FUNCTION_BLOCK FB_LoggerTest EXTENDS TcUnit.FB_TestSuite
VAR

END_VAR


T01_TestDodawaniaZgloszen ();
T02_TestDodawaniaZgloszen2 ();
T03_TestDodawaniaZgloszen3 ();

METHOD PRIVATE T01_TestDodawaniaZgloszen
VAR
	sttmpEvent: ST_BaseEvents_RowInQueue;
END_VAR
IF (TcUnit.TEST_ORDERED ('T01_TestDodawaniaZgloszen')) THEN
	WRITE_PROTECTED_BOOL (Ptr := ADR (GVL.fbLogger.bClearMemory), Value := TRUE);
	GVL.fbLogger ();
	AssertEquals_INT (Expected := 0, Actual := GVL.fbLogger.stBuffer.iNumerOfEvents, 	Message := 'T01a - bledna ilosc w kolejce');
	AssertEquals_INT (Expected := 0, Actual := GVL.fbLogger.stmemory.iNumberOfRow,		Message := 'T01b - bledna ilosc zgloszen');
//wyslanie zgloszenia 
	sttmpEvent.bActive				:= TRUE;
	sttmpEvent.bConfirm				:= TRUE;
	sttmpEvent.bIgnoreRepetitions	:= TRUE;
	sttmpEvent.dtStart				:= DT#2025-09-25-01:00:00;
	sttmpEvent.eEventCategory		:= E_BaseEvents_Category.Error;
	sttmpEvent.eEventAction			:= E_BaseEvents_Action.Start;
	sttmpEvent.uiIDEvent			:= 1;
	sttmpEvent.uiIDItem				:= 2;
	GVL.fbLogger.ReportEvent (stEvent := sttmpEvent);
	AssertEquals_INT (Expected := 1, Actual := GVL.fbLogger.stBuffer.iNumerOfEvents, 	Message := 'T02a - bledna ilosc w kolejce');
	AssertEquals_INT (Expected := 0, Actual := GVL.fbLogger.stmemory.iNumberOfRow,		Message := 'T02b - bledna ilosc zgloszen');
	GVL.fbLogger ();
	AssertEquals_INT (Expected := 0, Actual := GVL.fbLogger.stBuffer.iNumerOfEvents, 					Message := 'T03a - bledna ilosc w kolejce');
	AssertEquals_INT (Expected := 1, Actual := GVL.fbLogger.stmemory.iNumberOfRow,						Message := 'T03b - bledna ilosc zgloszen');
	AssertEquals_INT (Expected := 1, Actual := GVL.fbLogger.stNumberOfReports.iNumberOfActive,			Message := 'T03c - bledna ilosc zgloszen');
	AssertTrue (Condition := GVL.fbLogger.stNumberOfReports.arrActive [E_BaseEvents_Category.Error],	Message := 'T03d - bledny stan');
	AssertFalse (Condition := GVL.fbLogger.stNumberOfReports.arrActive [E_BaseEvents_Category.Alarm],	Message := 'T03d - bledny stan');
	AssertTrue (Condition := GVL.fbLogger.stNumberOfReports.bIsActive,									Message := 'T03e - bledny stan');
	AssertEquals_INT (Expected := 1, Actual := GVL.fbLogger.stNumberOfReports.iTotalNumer,				Message := 'T03f - bledna ilosc zgloszen');
//potwierdzenie zgloszenia 
	sttmpEvent.eEventAction			:= E_BaseEvents_Action.Confirm;
	sttmpEvent.uiIDEvent			:= 1;
	sttmpEvent.uiIDItem				:= 2;
	sttmpEvent.dtConfirmed			:= DT#2025-09-25-01:01:00;
	GVL.fbLogger.ReportEvent (stEvent := sttmpEvent);
	AssertEquals_INT (Expected := 1, Actual := GVL.fbLogger.stBuffer.iNumerOfEvents, 					Message := 'T04a - bledna ilosc w kolejce');
	AssertEquals_INT (Expected := 1, Actual := GVL.fbLogger.stmemory.iNumberOfRow,						Message := 'T04b - bledna ilosc zgloszen');
	GVL.fbLogger ();
	AssertEquals_INT (Expected := 0, Actual := GVL.fbLogger.stBuffer.iNumerOfEvents, 					Message := 'T05a - bledna ilosc w kolejce');
	AssertEquals_INT (Expected := 1, Actual := GVL.fbLogger.stmemory.iNumberOfRow,						Message := 'T05b - bledna ilosc zgloszen');
	AssertEquals_INT (Expected := 1, Actual := GVL.fbLogger.stNumberOfReports.iNumberOfActive,			Message := 'T05c - bledna ilosc zgloszen');
	AssertTrue (Condition := GVL.fbLogger.stNumberOfReports.arrActive [E_BaseEvents_Category.Error],	Message := 'T05d - bledny stan');
	AssertFalse (Condition := GVL.fbLogger.stNumberOfReports.arrActive [E_BaseEvents_Category.Alarm],	Message := 'T05d - bledny stan');
	AssertTrue (Condition := GVL.fbLogger.stNumberOfReports.bIsActive,									Message := 'T05e - bledny stan');
	AssertEquals_INT (Expected := 1, Actual := GVL.fbLogger.stNumberOfReports.iTotalNumer,				Message := 'T05f - bledna ilosc zgloszen');
//zamkniecie zgloszenia 
	sttmpEvent.eEventAction			:= E_BaseEvents_Action.Stop;
	sttmpEvent.uiIDEvent			:= 1;
	sttmpEvent.uiIDItem				:= 2;
	sttmpEvent.dtFinish				:= DT#2025-09-25-01:02:00;
	GVL.fbLogger.ReportEvent (stEvent := sttmpEvent);
	AssertEquals_INT (Expected := 1, Actual := GVL.fbLogger.stBuffer.iNumerOfEvents, 					Message := 'T04a - bledna ilosc w kolejce');
	AssertEquals_INT (Expected := 1, Actual := GVL.fbLogger.stmemory.iNumberOfRow,						Message := 'T04b - bledna ilosc zgloszen');
	GVL.fbLogger ();
	AssertEquals_INT (Expected := 0, Actual := GVL.fbLogger.stBuffer.iNumerOfEvents, 					Message := 'T05a - bledna ilosc w kolejce');
	AssertEquals_INT (Expected := 1, Actual := GVL.fbLogger.stmemory.iNumberOfRow,						Message := 'T05b - bledna ilosc zgloszen');
	AssertEquals_INT (Expected := 0, Actual := GVL.fbLogger.stNumberOfReports.iNumberOfActive,			Message := 'T05c - bledna ilosc zgloszen');
	AssertFalse (Condition := GVL.fbLogger.stNumberOfReports.arrActive [E_BaseEvents_Category.Error],	Message := 'T05d - bledny stan');
	AssertFalse (Condition := GVL.fbLogger.stNumberOfReports.arrActive [E_BaseEvents_Category.Alarm],	Message := 'T05d - bledny stan');
	Assertfalse (Condition := GVL.fbLogger.stNumberOfReports.bIsActive,									Message := 'T05e - bledny stan');
	AssertEquals_INT (Expected := 1, Actual := GVL.fbLogger.stNumberOfReports.iTotalNumer,				Message := 'T05f - bledna ilosc zgloszen');
	
	
	TcUnit.TEST_FINISHED ();
END_IF
END_METHOD

METHOD PRIVATE T02_TestDodawaniaZgloszen2
VAR
	sttmpEvent: ST_BaseEvents_RowInQueue;
END_VAR
IF (TcUnit.TEST_ORDERED ('T02_TestDodawaniaZgloszen2')) THEN
	GVL.fbLogger ();
	AssertEquals_INT (Expected := 0, Actual := GVL.fbLogger.stBuffer.iNumerOfEvents, 	Message := 'T01a - bledna ilosc w kolejce');
	AssertEquals_INT (Expected := 1, Actual := GVL.fbLogger.stmemory.iNumberOfRow,		Message := 'T01b - bledna ilosc zgloszen');
//wyslanie zgloszenia 
	sttmpEvent.bActive				:= TRUE;
	sttmpEvent.bConfirm				:= TRUE;
	sttmpEvent.bIgnoreRepetitions	:= TRUE;
	sttmpEvent.dtStart				:= DT#2025-09-25-02:00:00;
	sttmpEvent.eEventCategory		:= E_BaseEvents_Category.Error;
	sttmpEvent.eEventAction			:= E_BaseEvents_Action.Start;
	sttmpEvent.uiIDEvent			:= 1;
	sttmpEvent.uiIDItem				:= 2;
	GVL.fbLogger.ReportEvent (stEvent := sttmpEvent);
	AssertEquals_INT (Expected := 1, Actual := GVL.fbLogger.stBuffer.iNumerOfEvents, 					Message := 'T02a - bledna ilosc w kolejce');
	AssertEquals_INT (Expected := 1, Actual := GVL.fbLogger.stmemory.iNumberOfRow,						Message := 'T02b - bledna ilosc zgloszen');
	GVL.fbLogger ();
	AssertEquals_INT (Expected := 0, Actual := GVL.fbLogger.stBuffer.iNumerOfEvents, 					Message := 'T03a - bledna ilosc w kolejce');
	AssertEquals_INT (Expected := 2, Actual := GVL.fbLogger.stmemory.iNumberOfRow,						Message := 'T03b - bledna ilosc zgloszen');
	AssertEquals_INT (Expected := 1, Actual := GVL.fbLogger.stNumberOfReports.iNumberOfActive,			Message := 'T03c - bledna ilosc zgloszen');
	AssertTrue (Condition := GVL.fbLogger.stNumberOfReports.arrActive [E_BaseEvents_Category.Error],	Message := 'T03d - bledny stan');
	AssertFalse (Condition := GVL.fbLogger.stNumberOfReports.arrActive [E_BaseEvents_Category.Alarm],	Message := 'T03d - bledny stan');
	AssertTrue (Condition := GVL.fbLogger.stNumberOfReports.bIsActive,									Message := 'T03e - bledny stan');
	AssertEquals_INT (Expected := 2, Actual := GVL.fbLogger.stNumberOfReports.iTotalNumer,				Message := 'T03f - bledna ilosc zgloszen');
//zamkniecie zgloszenia  bez potwierdzenia a wymagane nic się nei powinno stać
	sttmpEvent.eEventAction			:= E_BaseEvents_Action.Stop;
	sttmpEvent.uiIDEvent			:= 1;
	sttmpEvent.uiIDItem				:= 2;
	sttmpEvent.dtFinish				:= DT#2025-09-25-02:00:00;
	GVL.fbLogger.ReportEvent (stEvent := sttmpEvent);
	AssertEquals_INT (Expected := 1, Actual := GVL.fbLogger.stBuffer.iNumerOfEvents, 					Message := 'T04a - bledna ilosc w kolejce');
	AssertEquals_INT (Expected := 2, Actual := GVL.fbLogger.stmemory.iNumberOfRow,						Message := 'T04b - bledna ilosc zgloszen');
	GVL.fbLogger ();
	AssertEquals_INT (Expected := 0, Actual := GVL.fbLogger.stBuffer.iNumerOfEvents, 					Message := 'T05a - bledna ilosc w kolejce');
	AssertEquals_INT (Expected := 2, Actual := GVL.fbLogger.stmemory.iNumberOfRow,						Message := 'T05b - bledna ilosc zgloszen');
	AssertEquals_INT (Expected := 1, Actual := GVL.fbLogger.stNumberOfReports.iNumberOfActive,			Message := 'T05c - bledna ilosc zgloszen');
	AssertTrue (Condition := GVL.fbLogger.stNumberOfReports.arrActive [E_BaseEvents_Category.Error],	Message := 'T05d - bledny stan');
	AssertFalse (Condition := GVL.fbLogger.stNumberOfReports.arrActive [E_BaseEvents_Category.Alarm],	Message := 'T05d - bledny stan');
	AssertTrue (Condition := GVL.fbLogger.stNumberOfReports.bIsActive,									Message := 'T05e - bledny stan');
	AssertEquals_INT (Expected := 2, Actual := GVL.fbLogger.stNumberOfReports.iTotalNumer,				Message := 'T05f - bledna ilosc zgloszen');
//potwierdzenie zgloszenia 
	sttmpEvent.eEventAction			:= E_BaseEvents_Action.Confirm;
	sttmpEvent.uiIDEvent			:= 1;
	sttmpEvent.uiIDItem				:= 2;
	sttmpEvent.dtConfirmed			:= DT#2025-09-25-02:01:00;
	GVL.fbLogger.ReportEvent (stEvent := sttmpEvent);
	AssertEquals_INT (Expected := 1, Actual := GVL.fbLogger.stBuffer.iNumerOfEvents, 					Message := 'T06a - bledna ilosc w kolejce');
	AssertEquals_INT (Expected := 2, Actual := GVL.fbLogger.stmemory.iNumberOfRow,						Message := 'T06b - bledna ilosc zgloszen');
	GVL.fbLogger ();
	AssertEquals_INT (Expected := 0, Actual := GVL.fbLogger.stBuffer.iNumerOfEvents, 					Message := 'T07a - bledna ilosc w kolejce');
	AssertEquals_INT (Expected := 2, Actual := GVL.fbLogger.stmemory.iNumberOfRow,						Message := 'T07b - bledna ilosc zgloszen');
	AssertEquals_INT (Expected := 1, Actual := GVL.fbLogger.stNumberOfReports.iNumberOfActive,			Message := 'T07c - bledna ilosc zgloszen');
	AssertTrue (Condition := GVL.fbLogger.stNumberOfReports.arrActive [E_BaseEvents_Category.Error],	Message := 'T07d - bledny stan');
	AssertFalse (Condition := GVL.fbLogger.stNumberOfReports.arrActive [E_BaseEvents_Category.Alarm],	Message := 'T07d - bledny stan');
	AssertTrue (Condition := GVL.fbLogger.stNumberOfReports.bIsActive,									Message := 'T07e - bledny stan');
	AssertEquals_INT (Expected := 2, Actual := GVL.fbLogger.stNumberOfReports.iTotalNumer,				Message := 'T07f - bledna ilosc zgloszen');
//zamkniecie zgloszenia 
	sttmpEvent.eEventAction			:= E_BaseEvents_Action.Stop;
	sttmpEvent.uiIDEvent			:= 1;
	sttmpEvent.uiIDItem				:= 2;
	sttmpEvent.dtFinish				:= DT#2025-09-25-02:02:00;
	GVL.fbLogger.ReportEvent (stEvent := sttmpEvent);
	AssertEquals_INT (Expected := 1, Actual := GVL.fbLogger.stBuffer.iNumerOfEvents, 					Message := 'T08a - bledna ilosc w kolejce');
	AssertEquals_INT (Expected := 2, Actual := GVL.fbLogger.stmemory.iNumberOfRow,						Message := 'T08b - bledna ilosc zgloszen');
	GVL.fbLogger ();
	AssertEquals_INT (Expected := 0, Actual := GVL.fbLogger.stBuffer.iNumerOfEvents, 					Message := 'T09a - bledna ilosc w kolejce');
	AssertEquals_INT (Expected := 2, Actual := GVL.fbLogger.stmemory.iNumberOfRow,						Message := 'T09b - bledna ilosc zgloszen');
	AssertEquals_INT (Expected := 0, Actual := GVL.fbLogger.stNumberOfReports.iNumberOfActive,			Message := 'T09c - bledna ilosc zgloszen');
	AssertFalse (Condition := GVL.fbLogger.stNumberOfReports.arrActive [E_BaseEvents_Category.Error],	Message := 'T09d - bledny stan');
	AssertFalse (Condition := GVL.fbLogger.stNumberOfReports.arrActive [E_BaseEvents_Category.Alarm],	Message := 'T09d - bledny stan');
	Assertfalse (Condition := GVL.fbLogger.stNumberOfReports.bIsActive,									Message := 'T09e - bledny stan');
	AssertEquals_INT (Expected := 2, Actual := GVL.fbLogger.stNumberOfReports.iTotalNumer,				Message := 'T09f - bledna ilosc zgloszen');
	
	
	TcUnit.TEST_FINISHED ();
END_IF
END_METHOD

METHOD PRIVATE T03_TestDodawaniaZgloszen3
VAR
	sttmpEvent: ST_BaseEvents_RowInQueue;
END_VAR
IF (TcUnit.TEST_ORDERED ('T03_TestDodawaniaZgloszen3')) THEN
//wyslanie zgloszenia 
	sttmpEvent.bActive				:= TRUE;
	sttmpEvent.bConfirm				:= FALSE;
	sttmpEvent.bIgnoreRepetitions	:= FALSE;
	sttmpEvent.dtStart				:= DT#2025-09-25-03:00:00;
	sttmpEvent.eEventCategory		:= E_BaseEvents_Category.Alarm;
	sttmpEvent.eEventAction			:= E_BaseEvents_Action.Start;
	sttmpEvent.uiIDEvent			:= 1;
	sttmpEvent.uiIDItem				:= 1;
	GVL.fbLogger.ReportEvent (stEvent := sttmpEvent);
	GVL.fbLogger ();
//zamkniecie zgloszenia 
	sttmpEvent.eEventAction			:= E_BaseEvents_Action.Stop;
	sttmpEvent.uiIDEvent			:= 1;
	sttmpEvent.uiIDItem				:= 1;
	sttmpEvent.dtFinish				:= DT#2025-09-25-03:02:00;
	GVL.fbLogger.ReportEvent (stEvent := sttmpEvent);
	GVL.fbLogger ();
//wyslanie zgloszenia 
	sttmpEvent.bActive				:= TRUE;
	sttmpEvent.bConfirm				:= FALSE;
	sttmpEvent.bIgnoreRepetitions	:= FALSE;
	sttmpEvent.dtStart				:= DT#2025-09-25-03:10:00;
	sttmpEvent.eEventCategory		:= E_BaseEvents_Category.Alarm;
	sttmpEvent.eEventAction			:= E_BaseEvents_Action.Start;
	sttmpEvent.uiIDEvent			:= 1;
	sttmpEvent.uiIDItem				:= 1;
	GVL.fbLogger.ReportEvent (stEvent := sttmpEvent);
	GVL.fbLogger ();
//wyslanie zgloszenia 
	sttmpEvent.bActive				:= TRUE;
	sttmpEvent.bConfirm				:= TRUE;
	sttmpEvent.bIgnoreRepetitions	:= TRUE;
	sttmpEvent.dtStart				:= DT#2025-09-25-03:20:00;
	sttmpEvent.eEventCategory		:= E_BaseEvents_Category.Error;
	sttmpEvent.eEventAction			:= E_BaseEvents_Action.Start;
	sttmpEvent.uiIDEvent			:= 2;
	sttmpEvent.uiIDItem				:= 1;
	GVL.fbLogger.ReportEvent (stEvent := sttmpEvent);
	GVL.fbLogger ();
//potwierdzenie zgloszenia 
	sttmpEvent.eEventAction			:= E_BaseEvents_Action.Confirm;
	sttmpEvent.uiIDEvent			:= 2;
	sttmpEvent.uiIDItem				:= 1;
	sttmpEvent.dtConfirmed			:= DT#2025-09-25-03:21:00;
	GVL.fbLogger.ReportEvent (stEvent := sttmpEvent);
	GVL.fbLogger ();
//zamkniecie zgloszenia 
	sttmpEvent.eEventAction			:= E_BaseEvents_Action.Stop;
	sttmpEvent.uiIDEvent			:= 2;
	sttmpEvent.uiIDItem				:= 1;
	sttmpEvent.dtFinish				:= DT#2025-09-25-03:22:00;
	GVL.fbLogger.ReportEvent (stEvent := sttmpEvent);
	GVL.fbLogger ();
//wyslanie zgloszenia 
	sttmpEvent.bActive				:= TRUE;
	sttmpEvent.bConfirm				:= FALSE;
	sttmpEvent.bIgnoreRepetitions	:= TRUE;
	sttmpEvent.dtStart				:= DT#2025-09-25-04:00:00;
	sttmpEvent.eEventCategory		:= E_BaseEvents_Category.Error;
	sttmpEvent.eEventAction			:= E_BaseEvents_Action.Start;
	sttmpEvent.uiIDEvent			:= 3;
	sttmpEvent.uiIDItem				:= 1;
	GVL.fbLogger.ReportEvent (stEvent := sttmpEvent);
	GVL.fbLogger ();
//wyslanie zgloszenia 
	sttmpEvent.bActive				:= TRUE;
	sttmpEvent.bConfirm				:= FALSE;
	sttmpEvent.bIgnoreRepetitions	:= TRUE;
	sttmpEvent.dtStart				:= DT#2025-09-25-04:20:00;
	sttmpEvent.eEventCategory		:= E_BaseEvents_Category.Message;
	sttmpEvent.eEventAction			:= E_BaseEvents_Action.Start;
	sttmpEvent.uiIDEvent			:= 4;
	sttmpEvent.uiIDItem				:= 1;
	GVL.fbLogger.ReportEvent (stEvent := sttmpEvent);
	GVL.fbLogger ();
//zamkniecie zgloszenia 
	sttmpEvent.eEventAction			:= E_BaseEvents_Action.Stop;
	sttmpEvent.uiIDEvent			:= 4;
	sttmpEvent.uiIDItem				:= 1;
	sttmpEvent.dtFinish				:= DT#2025-09-25-04:22:00;
	GVL.fbLogger.ReportEvent (stEvent := sttmpEvent);
	GVL.fbLogger ();
	
	
	TcUnit.TEST_FINISHED ();
END_IF
END_METHOD

END_FUNCTION_BLOCK

(* stored: Version 1.1.0.1, ProductVersion 3.1.4024.15
   POU FB_LoggerTest: Id {bdd902bd-8721-4963-bac8-ed229424c4e8}, SpecialFunc None
   Method T01_TestDodawaniaZgloszen: Id {95b1bee2-2fa2-40b4-ace9-9bed2d0ad664}
   Method T02_TestDodawaniaZgloszen2: Id {c6c2cab5-9412-4025-920f-725b656de169}
   Method T03_TestDodawaniaZgloszen3: Id {26235af6-606c-4534-abe3-d37bb2afacab} *)
